Fanuc TP program (LS listing): _sysvar_cfg.ls

/PROG  _SYSVAR_CFG
/ATTR
OWNER		= MNEDITOR;
COMMENT		= "Initial Setup";
PROG_SIZE	= 453;
CREATE		= DATE 23-10-27  TIME 05:42:28;
MODIFIED	= DATE 24-03-10  TIME 11:36:02;
FILE_NAME	= ;
VERSION		= 0;
LINE_COUNT	= 8;
MEMORY_SIZE	= 857;
PROTECT		= READ_WRITE;
TCD:  STACK_SIZE	= 0,
      TASK_PRIORITY	= 50,
      TIME_SLICE	= 0,
      BUSY_LAMP_OFF	= 0,
      ABORT_REQUEST	= 0,
      PAUSE_REQUEST	= 0;
DEFAULT_GROUP	= 1,*,*,*,*;
CONTROL_CODE	= 00000000 00000000;
LOCAL_REGISTERS	= 0,0,0;
/APPL

AUTO_SINGULARITY_HEADER;
  ENABLE_SINGULARITY_AVOIDANCE   : TRUE;
/MN
   1:  !******INIT SETUP-SYS VARS******* ;
   2:  $SCR.$COLDOVRD=25 ;
   3:  $SCR.$COORDOVRD=100 ;
   4:  $SCR.$TPENBLEOVRD=100 ;
   5:  $SCR.$FENCEOVRD=100 ;
   6:  $RGSPD_PREXE=1 ;
   7:  $RGTDB_PREXE=1 ;
   8:  $RGTRM_PREXE=1 ;
/POS
/END
